(* PLC project  *)

CONFIGURATION EK1100
END_CONFIGURATION
